{attribute 'GeneratedUsingTerminal: ER6002-0002-0022'}
{attribute addProperty BoxType "ER6002-0002-0022"}
{attribute addProperty Id "EtcSlaveTerminalBaseCOM_TxPDO_Map_Inputs_Channel_1AT %I*COM_TxPDO_Map_Inputs_Channel_6C2FC20224COM_TxPDO_Map_Inputs_Channel_2AT %I*COM_TxPDO_Map_Inputs_Channel_6C2FC20224COM_RxPDO_Map_Outputs_Channel_1AT %Q*COM_RxPDO_Map_Outputs_Channel_5D00B5E724COM_RxPDO_Map_Outputs_Channel_2AT %Q*COM_RxPDO_Map_Outputs_Channel_5D00B5E724WcStateAT %I*WcState_9091E0EB2InfoDataAT %I*InfoData_32EB74EA10"}
{attribute addProperty CRC "4006548345"}
{attribute addProperty Size "108"}
TYPE ER6002_EECF1379 EXTENDS EtcSlaveTerminalBase :
STRUCT
	{attribute addProperty Name "COM_TxPDO_Map_Inputs_Channel_1"}
	COM_TxPDO_Map_Inputs_Channel_1 : COM_TxPDO_Map_Inputs_Channel_6C2FC202;
	{attribute addProperty Name "COM_TxPDO_Map_Inputs_Channel_2"}
	COM_TxPDO_Map_Inputs_Channel_2 : COM_TxPDO_Map_Inputs_Channel_6C2FC202;
	{attribute addProperty Name "COM_RxPDO_Map_Outputs_Channel_1"}
	COM_RxPDO_Map_Outputs_Channel_1 : COM_RxPDO_Map_Outputs_Channel_5D00B5E7;
	{attribute addProperty Name "COM_RxPDO_Map_Outputs_Channel_2"}
	COM_RxPDO_Map_Outputs_Channel_2 : COM_RxPDO_Map_Outputs_Channel_5D00B5E7;
	{attribute addProperty Name "WcState"}
	WcState : WcState_9091E0EB;
	{attribute addProperty Name "InfoData"}
	InfoData : InfoData_32EB74EA;
END_STRUCT
END_TYPE

(* stored: Version 1.2.0.0, ProductVersion 3.1.4024.9
   DUT ER6002_EECF1379: Id {4c27d83a-9ac8-492a-b066-4df1d764cc1b} *)
